% RSLogix 500 project TESTING SCALING 1200 IF4_BAK003.RSS, saved by version 11.00.00.00 %
PROJECT "UNTITLED"    % processor: MicroLogix 1200 %

PROGRAM FILES
  LAD 2   6 rungs

DATA FILES
  O0 OUTPUT  4 elements
  I1 INPUT  11 elements
  S2 STATUS  66 elements
  B3 BINARY  1 elements
  T4 TIMER  1 elements
  C5 COUNTER  1 elements
  R6 CONTROL  1 elements
  N7 INTEGER  2 elements
  F8 FLOAT  1 elements

LADDER 2
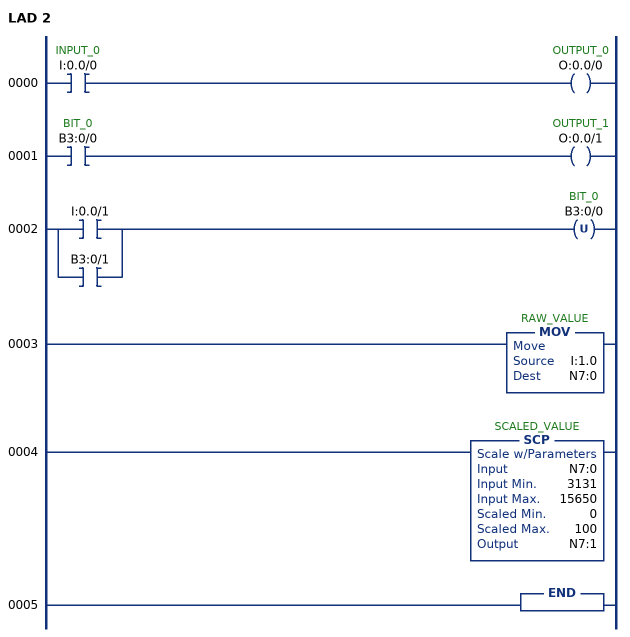
% Rung: 0 %
SOR XIC I:0.0/0 OTE O:0.0/0 EOR
%   I:0.0/0  INPUT_0 %
%   O:0.0/0  OUTPUT_0 %
% Rung: 1 %
SOR XIC B3:0/0 OTE O:0.0/1 EOR
%   B3:0/0  BIT_0 %
%   O:0.0/1  OUTPUT_1 %
% Rung: 2 %
SOR BST XIC I:0.0/1 NXB XIC B3:0/1 BND OTU B3:0/0 EOR
%   B3:0/0  BIT_0 %
% Rung: 3 %
SOR MOV I:1.0 N7:0 EOR
%   N7:0  RAW_VALUE %
% Rung: 4 %
SOR SCP N7:0 3131 15650 0 100 N7:1 EOR
%   N7:0  RAW_VALUE %
%   N7:1  SCALED_VALUE %
% Rung: 5 %
SOR END EOR

OTHER DOCUMENTED ADDRESSES
  I:1.0/0  FLOAT
  INPUT_1  
